// TIA Portal V21 export
TYPE "LAxisCtrl_typeAxisConfig"
TITLE = LAxisCtrl_typeAxisConfig
// Support: tech.team.motioncontrol@siemens.com
   STRUCT
      generalSettings : "LAxisCtrl_typeGeneralSettings";   // Configuration of general settings
      power : "LAxisCtrl_typePower";   // Configuration of MC_POWER function
      jog : "LAxisCtrl_typeJog";   // Configuration of JOG function
      moveVelocity : "LAxisCtrl_typeMoveVelocity";   // Configuration of MC_MOVEVELOCITY function
      stop : "LAxisCtrl_typeStop";   // Configuration of MC_HALT function
      fastStop : "LAxisCtrl_typeFastStop";   // Configuration of MC_HALT function (alternative dynamics)
      torqueLimiting : "LAxisCtrl_typeTorqueLimiting";   // Configuration of MC_TORQUELIMITING function
      homing : "LAxisCtrl_typeHoming";   // Configuration of HOMING function
      posRelative : "LAxisCtrl_typePosRelative";   // Configuration of MC_MOVERELATIVE function
      posAbsolute : "LAxisCtrl_typePosAbsolute";   // Configuration of MC_MOVEABSOLUTE function
      posSuperimposed : "LAxisCtrl_typePosSuperimposed";   // Configuration of MC_MOVESUPERIMPOSED function
      haltSuperimposed : "LAxisCtrl_typeHaltSuperimposed";   // Configuration of MC_HALTSUPERIMPOSED function
      gearInRelative : "LAxisCtrl_typeGearInRelative";   // Configuration of MC_GEARIN function
      gearInAbsolute : "LAxisCtrl_typeGearInAbsolute";   // Configuration of MC_GEARIN_POS function
      gearInVelocity : "LAxisCtrl_typeGearInVelocity";   // Configuration of MC_GEARINVELOCITY function
      camIn : "LAxisCtrl_typeCamIn";   // Configuration of MC_CAMIN function
      gearOutCamOut : "LAxisCtrl_typeGearOutCamOut";   // Configuration of MC_GEAROUT / MC_CAMOUT function
      phasing : "LAxisCtrl_typePhasing";   // Configuration of MC_PHASING function
      offset : "LAxisCtrl_typeOffset";   // Configuration of MC_OFFSET function
   END_STRUCT;
END_TYPE
